Yaskawa INFORM job: B-7-08279-80-90-R.JBI

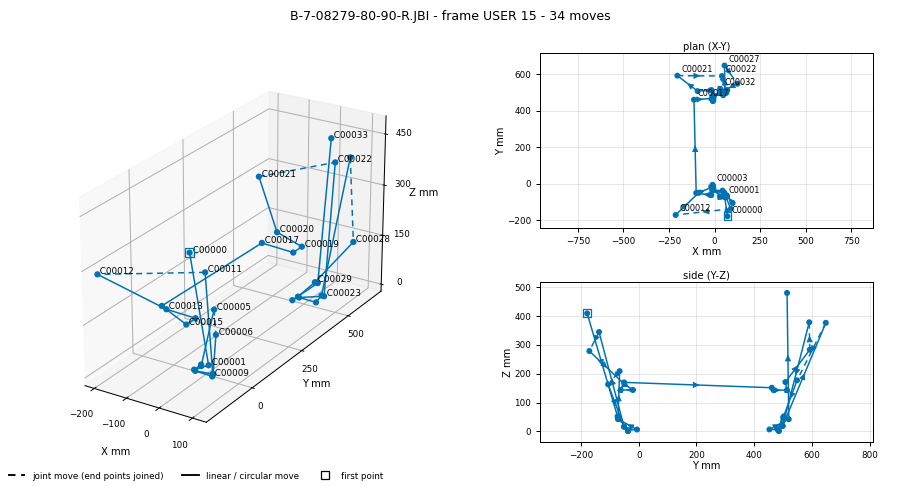
[picture p0: tool path of B-7-08279-80-90-R.JBI in frame USER 15, 34 of 34 moves have a stored position in this frame; points joined in program order, loops and branches not executed]
/JOB
//NAME B-7-08279-80-90-R
///FOLDERNAME PART_420-08279-80
//POS
///NPOS 34,0,34,0,0,0
///USER 15
///TOOL 4
///POSTYPE USER
///RECTAN
///RCONF 1,0,0,0,0,0,0,0,0,0,0,0,0,0,0,0,0,0,0,0,0,0,0,0
C00000=70.970,-178.868,409.213,-165.0000,45.0000,0.0000
C00001=55.971,-73.592,51.975,-165.0011,45.0003,0.0032
C00002=-12.407,-36.914,4.666,-178.0423,55.7437,-36.8725
C00003=-10.903,-5.926,6.493,-178.0437,55.7456,-36.8764
C00004=32.283,-72.150,42.455,-165.0000,45.0000,0.0000
C00005=68.685,-66.272,209.042,-165.0000,45.0000,0.0000
C00006=99.538,-106.298,163.160,-166.3780,45.3490,-50.4350
C00007=54.885,-50.957,16.272,155.8958,41.5580,-103.2447
C00008=-8.888,-36.814,2.198,130.3659,26.1559,-138.9484
C00009=43.660,-37.448,0.781,130.3624,26.1599,-138.9477
C00010=53.929,-50.980,16.227,147.3699,35.8055,-116.8283
C00011=88.912,-137.678,344.705,-160.0731,43.4104,-40.2210
C00012=-213.482,-171.326,278.744,154.4200,34.7310,45.4810
C00013=-87.212,-49.799,163.694,107.6090,9.3560,77.2190
C00014=-17.646,-19.929,143.778,104.0913,8.5645,76.6652
C00015=-17.856,-62.779,143.481,104.0933,8.5652,76.6629
C00016=-100.598,-50.810,170.079,107.6090,9.3560,77.2190
C00017=-112.794,461.129,151.518,107.5190,-7.4490,103.3910
C00018=-16.463,467.682,143.004,97.5717,-4.9492,104.4453
C00019=-16.348,513.716,143.272,97.5722,-4.9507,104.4466
C00020=-92.930,508.215,171.083,107.5190,-7.4490,103.3910
C00021=-203.967,592.873,283.205,107.5190,-7.4490,103.3910
C00022=40.454,590.981,378.479,-169.5230,46.0050,83.6620
C00023=64.926,498.805,18.936,-133.5620,7.6410,152.0390
C00024=-6.974,485.685,2.315,-128.5831,10.2499,151.3320
C00025=47.348,485.481,1.282,-128.5832,10.2490,151.3370
C00026=56.860,498.850,19.061,-133.5613,7.6425,152.0382
C00027=54.868,648.552,376.545,-169.5230,46.0050,83.6620
C00028=125.357,548.743,177.335,165.0000,45.0000,0.0000
C00029=33.224,502.241,52.156,165.0000,45.0000,0.0000
C00030=-7.749,481.182,6.767,165.0871,51.2780,6.9835
C00031=-8.939,452.916,6.812,160.5522,52.5763,15.9587
C00032=32.283,520.083,42.455,165.0000,45.0000,0.0000
C00033=70.181,514.089,480.075,165.0008,44.9999,-0.0009
///POSTYPE ANGLE
///ANGLE
EC00000=90.0000
///TOOL 0
EC00001=90.0000
EC00002=90.0000
EC00003=90.0000
///TOOL 4
EC00004=90.0000
EC00005=90.0000
EC00006=105.0000
///TOOL 0
EC00007=105.0000
EC00008=105.0000
EC00009=105.0000
EC00010=105.0000
EC00011=105.0000
///TOOL 4
EC00012=135.0000
EC00013=135.0000
///TOOL 0
EC00014=135.0000
EC00015=135.0000
///TOOL 4
EC00016=135.0000
EC00017=135.0000
///TOOL 0
EC00018=135.0000
EC00019=135.0000
///TOOL 4
EC00020=135.0000
EC00021=135.0000
EC00022=105.0000
EC00023=105.0000
///TOOL 0
EC00024=105.0000
EC00025=105.0000
EC00026=105.0000
///TOOL 4
EC00027=105.0000
EC00028=90.0000
EC00029=90.0000
///TOOL 0
EC00030=90.0000
EC00031=90.0000
///TOOL 4
EC00032=90.0000
///TOOL 0
EC00033=90.0000
//INST
///DATE 2021/10/29 11:36
///ATTR SC,RW,RJ
////FRAME USER 15
///GROUP1 RB1
///GROUP2 ST3
NOP
'Path Start: PP1_1
MOVJ C00000 VJ=100.00  +MOVJ EC00000
SMOVL C00001 V=1250.0  +MOVJ EC00001
SMOVL C00002 V=1250.0  +MOVJ EC00002
ARCON ASF#(951)
SMOVL C00003 V=8.5  +MOVJ EC00003
ARCOF AEF#(951)
SMOVL C00004 V=1250.0  +MOVJ EC00004
SMOVL C00005 V=1250.0  +MOVJ EC00005
'Path End
'Path Start: PP48
MOVJ C00006 VJ=100.00  +MOVJ EC00006
SMOVL C00007 V=1250.0  +MOVJ EC00007
SMOVL C00008 V=300.0  +MOVJ EC00008
ARCON ASF#(953)
SMOVL C00009 V=15.7  +MOVJ EC00009
ARCOF AEF#(953)
SMOVL C00010 V=1250.0  +MOVJ EC00010
SMOVL C00011 V=1250.0  +MOVJ EC00011
'Path End
'Path Start: PP47
MOVJ C00012 VJ=100.00  +MOVJ EC00012
SMOVL C00013 V=1250.0  +MOVJ EC00013
SMOVL C00014 V=300.0  +MOVJ EC00014
ARCON ASF#(953)
SMOVL C00015 V=12.7  +MOVJ EC00015
ARCOF AEF#(953)
SMOVL C00016 V=1250.0  +MOVJ EC00016
'Path End
'Path Start: PP42
SMOVL C00017 V=1250.0  +MOVJ EC00017
SMOVL C00018 V=300.0  +MOVJ EC00018
ARCON ASF#(953)
SMOVL C00019 V=12.7  +MOVJ EC00019
ARCOF AEF#(953)
SMOVL C00020 V=1250.0  +MOVJ EC00020
SMOVL C00021 V=1250.0  +MOVJ EC00021
'Path End
'Path Start: PP41
MOVJ C00022 VJ=100.00  +MOVJ EC00022
SMOVL C00023 V=1250.0  +MOVJ EC00023
SMOVL C00024 V=300.0  +MOVJ EC00024
ARCON ASF#(953)
SMOVL C00025 V=15.7  +MOVJ EC00025
ARCOF AEF#(953)
SMOVL C00026 V=1250.0  +MOVJ EC00026
SMOVL C00027 V=1250.0  +MOVJ EC00027
'Path End
'Path Start: PP1
MOVJ C00028 VJ=100.00  +MOVJ EC00028
SMOVL C00029 V=1250.0  +MOVJ EC00029
SMOVL C00030 V=1250.0  +MOVJ EC00030
ARCON ASF#(951)
SMOVL C00031 V=8.5  +MOVJ EC00031
ARCOF AEF#(951)
SMOVL C00032 V=1250.0  +MOVJ EC00032
SMOVL C00033 V=1250.0  +MOVJ EC00033
INC I005
'Path End
END
